KUKA KRL program: Station200_UpStacker.src, Station200_UpStacker.dat

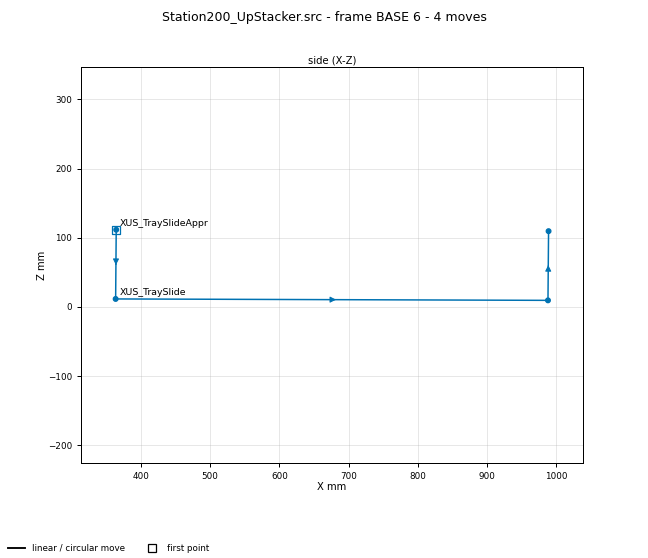
[picture p0: tool path of Station200_UpStacker.src in frame BASE 6, 4 of 12 moves have a stored position in this frame; points joined in program order, loops and branches not executed]
--- Station200_UpStacker.src ---
&ACCESS RVO1
&REL 54
&PARAM DISKPATH = KRC:\R1\Program
DEF Station200_UpStacker()

   ;FOLD INI;%{PE}
      ;FOLD BASISTECH INI
         GLOBAL INTERRUPT DECL 3 WHEN $STOPMESS == TRUE DO IR_STOPM()
         INTERRUPT ON 3
         BAS(#INITMOV, 0)
      ;ENDFOLD (BASISTECH INI)
      ;FOLD USER INI
         ;Make your modifications here
      ;ENDFOLD (USER INI)
      ;ENDFOLD (INI)

      PickPlaceTrayTeach()

;FOLD SPTP US_A1Turn Vel=100 % PDAT8 Tool[0] Base[0] ;%{PE}
;FOLD Parameters ;%{h}
;Params IlfProvider=kukaroboter.basistech.inlineforms.movement.spline; Kuka.IsGlobalPoint=False; Kuka.PointName=US_A1Turn; Kuka.BlendingEnabled=False; Kuka.MoveDataPtpName=PDAT8; Kuka.VelocityPtp=100; Kuka.VelocityFieldEnabled=True; Kuka.ColDetectFieldEnabled=True; Kuka.CurrentCDSetIndex=0; Kuka.MovementParameterFieldEnabled=True; IlfCommand=SPTP
;ENDFOLD
SPTP XUS_A1Turn WITH $VEL_AXIS[1] = SVEL_JOINT(100.0), $TOOL = STOOL2(FUS_A1Turn), $BASE = SBASE(FUS_A1Turn.BASE_NO), $IPO_MODE = SIPO_MODE(FUS_A1Turn.IPO_FRAME), $LOAD = SLOAD(FUS_A1Turn.TOOL_NO), $ACC_AXIS[1] = SACC_JOINT(PPDAT8), $APO = SAPO_PTP(PPDAT8), $GEAR_JERK[1] = SGEAR_JERK(PPDAT8), $COLLMON_TOL_PRO[1] = USE_CM_PRO_VALUES(0)
;ENDFOLD

;If tray layer needs to be moved, move layer before anything else happens.
If UStoR_ReqToMoveLayer==True Then
;FOLD SPTP US_TraySlideAppr Vel=100 % PDAT9 Tool[3]:TraySlidePin Base[6]:StackerFrame ;%{PE}
;FOLD Parameters ;%{h}
;Params IlfProvider=kukaroboter.basistech.inlineforms.movement.spline; Kuka.IsGlobalPoint=False; Kuka.PointName=US_TraySlideAppr; Kuka.BlendingEnabled=False; Kuka.MoveDataPtpName=PDAT9; Kuka.VelocityPtp=100; Kuka.VelocityFieldEnabled=True; Kuka.ColDetectFieldEnabled=True; Kuka.CurrentCDSetIndex=0; Kuka.MovementParameterFieldEnabled=True; IlfCommand=SPTP
;ENDFOLD
SPTP XUS_TraySlideAppr WITH $VEL_AXIS[1] = SVEL_JOINT(100.0), $TOOL = STOOL2(FUS_TraySlideAppr), $BASE = SBASE(FUS_TraySlideAppr.BASE_NO), $IPO_MODE = SIPO_MODE(FUS_TraySlideAppr.IPO_FRAME), $LOAD = SLOAD(FUS_TraySlideAppr.TOOL_NO), $ACC_AXIS[1] = SACC_JOINT(PPDAT9), $APO = SAPO_PTP(PPDAT9), $GEAR_JERK[1] = SGEAR_JERK(PPDAT9), $COLLMON_TOL_PRO[1] = USE_CM_PRO_VALUES(0)
;ENDFOLD
;FOLD SLIN US_TraySlide Vel=0.2 m/s CPDAT07 Tool[3]:TraySlidePin Base[6]:StackerFrame ;%{PE}
;FOLD Parameters ;%{h}
;Params IlfProvider=kukaroboter.basistech.inlineforms.movement.spline; Kuka.IsGlobalPoint=False; Kuka.PointName=US_TraySlide; Kuka.BlendingEnabled=False; Kuka.MoveDataName=CPDAT07; Kuka.VelocityPath=0.2; Kuka.VelocityFieldEnabled=True; Kuka.ColDetectFieldEnabled=True; Kuka.CurrentCDSetIndex=0; Kuka.MovementParameterFieldEnabled=True; IlfCommand=SLIN
;ENDFOLD
SLIN XUS_TraySlide WITH $VEL = SVEL_CP(0.2, , LCPDAT07), $TOOL = STOOL2(FUS_TraySlide), $BASE = SBASE(FUS_TraySlide.BASE_NO), $IPO_MODE = SIPO_MODE(FUS_TraySlide.IPO_FRAME), $LOAD = SLOAD(FUS_TraySlide.TOOL_NO), $ACC = SACC_CP(LCPDAT07), $ORI_TYPE = SORI_TYP(LCPDAT07), $APO = SAPO(LCPDAT07), $JERK = SJERK(LCPDAT07), $COLLMON_TOL_PRO[1] = USE_CM_PRO_VALUES(0)
;ENDFOLD
;FOLD SLIN US_TraySlideEnd Vel=0.15 m/s CPDAT08 Tool[3]:TraySlidePin Base[6]:StackerFrame ;%{PE}
;FOLD Parameters ;%{h}
;Params IlfProvider=kukaroboter.basistech.inlineforms.movement.spline; Kuka.IsGlobalPoint=False; Kuka.PointName=US_TraySlideEnd; Kuka.BlendingEnabled=False; Kuka.MoveDataName=CPDAT08; Kuka.VelocityPath=0.15; Kuka.VelocityFieldEnabled=True; Kuka.ColDetectFieldEnabled=True; Kuka.CurrentCDSetIndex=0; Kuka.MovementParameterFieldEnabled=True; IlfCommand=SLIN
;ENDFOLD
SLIN XUS_TraySlideEnd WITH $VEL = SVEL_CP(0.15, , LCPDAT08), $TOOL = STOOL2(FUS_TraySlideEnd), $BASE = SBASE(FUS_TraySlideEnd.BASE_NO), $IPO_MODE = SIPO_MODE(FUS_TraySlideEnd.IPO_FRAME), $LOAD = SLOAD(FUS_TraySlideEnd.TOOL_NO), $ACC = SACC_CP(LCPDAT08), $ORI_TYPE = SORI_TYP(LCPDAT08), $APO = SAPO(LCPDAT08), $JERK = SJERK(LCPDAT08), $COLLMON_TOL_PRO[1] = USE_CM_PRO_VALUES(0)
;ENDFOLD
;FOLD SLIN US_TraySlideReturn Vel=0.2 m/s CPDAT09 Tool[3]:TraySlidePin Base[6]:StackerFrame ;%{PE}
;FOLD Parameters ;%{h}
;Params IlfProvider=kukaroboter.basistech.inlineforms.movement.spline; Kuka.IsGlobalPoint=False; Kuka.PointName=US_TraySlideReturn; Kuka.BlendingEnabled=False; Kuka.MoveDataName=CPDAT09; Kuka.VelocityPath=0.2; Kuka.VelocityFieldEnabled=True; Kuka.ColDetectFieldEnabled=True; Kuka.CurrentCDSetIndex=0; Kuka.MovementParameterFieldEnabled=True; IlfCommand=SLIN
;ENDFOLD
SLIN XUS_TraySlideReturn WITH $VEL = SVEL_CP(0.2, , LCPDAT09), $TOOL = STOOL2(FUS_TraySlideReturn), $BASE = SBASE(FUS_TraySlideReturn.BASE_NO), $IPO_MODE = SIPO_MODE(FUS_TraySlideReturn.IPO_FRAME), $LOAD = SLOAD(FUS_TraySlideReturn.TOOL_NO), $ACC = SACC_CP(LCPDAT09), $ORI_TYPE = SORI_TYP(LCPDAT09), $APO = SAPO(LCPDAT09), $JERK = SJERK(LCPDAT09), $COLLMON_TOL_PRO[1] = USE_CM_PRO_VALUES(0)
;ENDFOLD
;FOLD SPTP DS_A1Turn Vel=100 % PDAT10 Tool[0] Base[0] ;%{PE}
;FOLD Parameters ;%{h}
;Params IlfProvider=kukaroboter.basistech.inlineforms.movement.spline; Kuka.IsGlobalPoint=False; Kuka.PointName=DS_A1Turn; Kuka.BlendingEnabled=False; Kuka.MoveDataPtpName=PDAT10; Kuka.VelocityPtp=100; Kuka.VelocityFieldEnabled=True; Kuka.ColDetectFieldEnabled=True; Kuka.CurrentCDSetIndex=0; Kuka.MovementParameterFieldEnabled=True; IlfCommand=SPTP
;ENDFOLD
SPTP XDS_A1Turn WITH $VEL_AXIS[1] = SVEL_JOINT(100.0), $TOOL = STOOL2(FDS_A1Turn), $BASE = SBASE(FDS_A1Turn.BASE_NO), $IPO_MODE = SIPO_MODE(FDS_A1Turn.IPO_FRAME), $LOAD = SLOAD(FDS_A1Turn.TOOL_NO), $ACC_AXIS[1] = SACC_JOINT(PPDAT10), $APO = SAPO_PTP(PPDAT10), $GEAR_JERK[1] = SGEAR_JERK(PPDAT10), $COLLMON_TOL_PRO[1] = USE_CM_PRO_VALUES(0)
;ENDFOLD
       RtoUS_LayerMovedConfirm=True
       wait sec .1
       RtoUS_LayerMovedConfirm=False
GOTO EndOfModule
EndIf


;Clear vacuum cups outputs
RtoPLC_BlankCupAVac=False
RtoPLC_BlankCupBVac=False
RtoPLC_BlankCupABlow=False
RtoPLC_BlankCupBBlow=False
RtoUS_PickConfirm=False
RobotCell_Error=False

;Check for layer mover, if needed slide upstacker tray to downstacker



 ;move tooling to row and column approach position for pick, then slowy move into the pick position
            US_PickApproach[UStoR_PickRowNumber,UStoR_PickColumnNumber] = US_Pick[UStoR_PickRowNumber,UStoR_PickColumnNumber]
            US_PickApproach[UStoR_PickRowNumber,UStoR_PickColumnNumber].Z = US_PickApproach[UStoR_PickRowNumber,UStoR_PickColumnNumber].Z + 100
            US_PickApproachSlow[UStoR_PickRowNumber,UStoR_PickColumnNumber].Z = US_PickApproach[UStoR_PickRowNumber,UStoR_PickColumnNumber].Z - 65


 SPTP US_PickApproach[UStoR_PickRowNumber,UStoR_PickColumnNumber] with $TOOL=TOOL_DATA[1],$BASE=BASE_DATA[1],$LOAD=LOAD_DATA[1],$VEL.CP = 2
 SLIN US_PickApproachSlow[UStoR_PickRowNumber,UStoR_PickColumnNumber] with $TOOL=TOOL_DATA[1],$BASE=BASE_DATA[1],$LOAD=LOAD_DATA[1],$VEL.CP = 2
 SLIN US_Pick[UStoR_PickRowNumber,UStoR_PickColumnNumber] with $TOOL=TOOL_DATA[1],$BASE=BASE_DATA[1],$LOAD=LOAD_DATA[1],$VEL.CP = 0.1

;Set vacuum cups to on
RtoPLC_BlankCupAVac=True
RtoPLC_BlankCupBVac=True

      $TIMER_STOP[2]=True ;stop timer
       $TIMER[2]=0 ;reset timer
       $TIMER_STOP[2]=False ;stop timer
       Loop
       If (($TIMER[2]>=5000) Or ((PLCtoR_BlankCupAVacOn==True) And (PLCtoR_BlankCupBVacOn==True)))Then
              $TIMER_STOP[2]=True ;stop timer
              $TIMER[2]=0 ;reset time
             Exit
endif
         EndLoop
;check vacuum sensors for being false, if false, set suction cup error bits
If ((PLCtoR_BlankCupAVacOn==False) Or (PLCtoR_BlankCupBVacOn==False)) Then

       If PLCtoR_BlankCupAVacOn==False Then
              RtoUS_PickErrorVG524=True

       EndIf
       If PLCtoR_BlankCupBVacOn==False Then
              RtoUS_PickErrorVG526=True

       EndIf
EndIf

;check if vacuum error bits were set, if set, turn off vacuum cups, blow off, reset error bits
If ((RtoUS_PickErrorVG524==True) Or (RtoUS_PickErrorVG526==True)) Then
       Wait Sec .25
       RtoPLC_BlankCupAVac=False
       RtoPLC_BlankCupBVac=False
       RtoPLC_BlankCupABlow=True
       RtoPLC_BlankCupBBlow=True
       Wait Sec .25
       RtoPLC_BlankCupABlow=False
       RtoPLC_BlankCupBBlow=False
       RtoUS_PickErrorVG524=False
       RtoUS_PickErrorVG526=False

       SLIN US_PickApproach[UStoR_PickRowNumber,UStoR_PickColumnNumber] with $TOOL=TOOL_DATA[1],$BASE=BASE_DATA[1],$LOAD=LOAD_DATA[1],$VEL.CP = 2
EndIf

;check vacuum sensors for being true, if true, slowly lift parts from tray
If ((PLCtoR_BlankCupAVacOn==True) And (PLCtoR_BlankCupBVacOn==True)) Then
       SLIN US_PickApproach[UStoR_PickRowNumber,UStoR_PickColumnNumber] with $TOOL=TOOL_DATA[1],$BASE=BASE_DATA[1],$LOAD=LOAD_DATA[1],$VEL.CP = 2
EndIf


;FOLD SPTP US_A1Return Vel=100 % PDAT4 Tool[0] Base[0] ;%{PE}
;FOLD Parameters ;%{h}
;Params IlfProvider=kukaroboter.basistech.inlineforms.movement.spline; Kuka.IsGlobalPoint=False; Kuka.PointName=US_A1Return; Kuka.BlendingEnabled=False; Kuka.MoveDataPtpName=PDAT4; Kuka.VelocityPtp=100; Kuka.VelocityFieldEnabled=True; Kuka.ColDetectFieldEnabled=True; Kuka.CurrentCDSetIndex=0; Kuka.MovementParameterFieldEnabled=True; IlfCommand=SPTP
;ENDFOLD
SPTP XUS_A1Return WITH $VEL_AXIS[1] = SVEL_JOINT(100.0), $TOOL = STOOL2(FUS_A1Return), $BASE = SBASE(FUS_A1Return.BASE_NO), $IPO_MODE = SIPO_MODE(FUS_A1Return.IPO_FRAME), $LOAD = SLOAD(FUS_A1Return.TOOL_NO), $ACC_AXIS[1] = SACC_JOINT(PPDAT4), $APO = SAPO_PTP(PPDAT4), $GEAR_JERK[1] = SGEAR_JERK(PPDAT4), $COLLMON_TOL_PRO[1] = USE_CM_PRO_VALUES(0)
;ENDFOLD

;check vacuum sensors again for being false, if false, set suction cup error bits
If ((PLCtoR_BlankCupAVacOn==False) Or (PLCtoR_BlankCupBVacOn==False)) Then
       Wait Sec 2
       If PLCtoR_BlankCupAVacOn==False Then
              RtoUS_PickErrorVG524=True

       EndIf
       If PLCtoR_BlankCupBVacOn==False Then
              RtoUS_PickErrorVG526=True

       EndIf
EndIf

;check vacuum sensors again for being true, if true, set pick confirm bit for .5 seconds, copy sequence number to tool, set tooling has-parts bit,  END this module program
If ((PLCtoR_BlankCupAVacOn==True) And (PLCtoR_BlankCupBVacOn==True)) Then
       RtoPLC_ToolBlnkSeqNumber=UStoR_PickSeqNumber
       RtoUS_PickConfirm=True
       Wait Sec .25
       RtoUS_PickConfirm=False
       RtoPLC_ToolBlnkHasParts=True

EndIf

;check again if vacuum error bits were set, if set, turn off vacuum cups, blow off, reset error bits, set tooling has-parts bit, call reject blanks module program
If ((RtoUS_PickErrorVG524==True) Or (RtoUS_PickErrorVG526==True)) Then
       Wait Sec .25
       RtoUS_PickErrorVG524=False
       RtoUS_PickErrorVG526=False
       RtoPLC_ToolBlnkHasParts=True
       Rjct_1Blnk_2Fin_3Both=1
       Station500_Reject()
EndIf


EndOfModule:
END

--- Station200_UpStacker.dat ---
&ACCESS RVP1
&REL 55
&PARAM DISKPATH = KRC:\R1\Program
DEFDAT  STATION200_UPSTACKER
;FOLD EXTERNAL DECLARATIONS;%{PE}%MKUKATPBASIS,%CEXT,%VCOMMON,%P
;FOLD BASISTECH EXT;%{PE}%MKUKATPBASIS,%CEXT,%VEXT,%P
EXT  BAS (BAS_COMMAND  :IN,REAL  :IN )
DECL INT SUCCESS
;ENDFOLD (BASISTECH EXT)
;FOLD USER EXT;%{E}%MKUKATPUSER,%CEXT,%VEXT,%P
;Make your modifications here

;ENDFOLD (USER EXT)
;ENDFOLD (EXTERNAL DECLARATIONS)


DECL LDAT LCPDAT1={VEL 2.00000,ACC 60.0000,APO_DIST 500.000,APO_FAC 50.0000,AXIS_VEL 100.000,AXIS_ACC 60.0000,ORI_TYP #VAR,CIRC_TYP #BASE,JERK_FAC 50.0000,GEAR_JERK 100.000,EXAX_IGN 0}
DECL PDAT PDEFAULT={VEL 100.000,ACC 60.0000,APO_DIST 500.000,APO_MODE #CDIS,GEAR_JERK 100.000,EXAX_IGN 0}
DECL LDAT LCPDAT2={VEL 2.00000,ACC 60.0000,APO_DIST 500.000,APO_FAC 50.0000,AXIS_VEL 100.000,AXIS_ACC 60.0000,ORI_TYP #VAR,CIRC_TYP #BASE,JERK_FAC 50.0000,GEAR_JERK 100.000,EXAX_IGN 0}
DECL PDAT PPDAT1={VEL 100.000,ACC 60.0000,APO_DIST 500.000,APO_MODE #CDIS,GEAR_JERK 100.000,EXAX_IGN 0}
DECL LDAT LCPDAT3={VEL 2.00000,ACC 60.0000,APO_DIST 500.000,APO_FAC 50.0000,AXIS_VEL 100.000,AXIS_ACC 60.0000,ORI_TYP #VAR,CIRC_TYP #BASE,JERK_FAC 50.0000,GEAR_JERK 100.000,EXAX_IGN 0}
DECL LDAT LCPDAT4={VEL 2.00000,ACC 60.0000,APO_DIST 500.000,APO_FAC 50.0000,AXIS_VEL 100.000,AXIS_ACC 60.0000,ORI_TYP #VAR,CIRC_TYP #BASE,JERK_FAC 50.0000,GEAR_JERK 100.000,EXAX_IGN 0}
DECL LDAT LCPDAT5={VEL 2.00000,ACC 60.0000,APO_DIST 500.000,APO_FAC 50.0000,AXIS_VEL 100.000,AXIS_ACC 60.0000,ORI_TYP #VAR,CIRC_TYP #BASE,JERK_FAC 50.0000,GEAR_JERK 100.000,EXAX_IGN 0}
DECL PDAT PPDAT2={VEL 100.000,ACC 60.0000,APO_DIST 500.000,APO_MODE #CDIS,GEAR_JERK 100.000,EXAX_IGN 0}
DECL PDAT PPDAT3={VEL 100.000,ACC 60.0000,APO_DIST 500.000,APO_MODE #CDIS,GEAR_JERK 100.000,EXAX_IGN 0}
DECL PDAT PPDAT4={VEL 100.000,ACC 60.0000,APO_DIST 500.000,APO_MODE #CDIS,GEAR_JERK 100.000,EXAX_IGN 0}
DECL E6POS XUS_A1Turn={X -108.546844,Y -232.779465,Z 1087.90991,A 64.9999619,B 35.0000,C 179.999985,S 2,T 34,E1 0.0,E2 0.0,E3 0.0,E4 0.0,E5 0.0,E6 0.0}
DECL FDAT FUS_A1Turn={TOOL_NO 0,BASE_NO 0,IPO_FRAME #BASE,POINT2[] " "}
DECL E6POS XUS_A1Return={X -108.546844,Y -232.779465,Z 1087.90991,A 64.9999619,B 35.0000,C 179.999985,S 2,T 34,E1 0.0,E2 0.0,E3 0.0,E4 0.0,E5 0.0,E6 0.0}
DECL FDAT FUS_A1Return={TOOL_NO 0,BASE_NO 0,IPO_FRAME #BASE,POINT2[] " "}
DECL LDAT LCPDAT6={VEL 2.00000,ACC 60.0000,APO_DIST 500.000,APO_FAC 50.0000,AXIS_VEL 100.000,AXIS_ACC 60.0000,ORI_TYP #VAR,CIRC_TYP #BASE,JERK_FAC 50.0000,GEAR_JERK 100.000,EXAX_IGN 0}
DECL LDAT LCPDAT7={VEL 2.00000,ACC 60.0000,APO_DIST 500.000,APO_FAC 50.0000,AXIS_VEL 100.000,AXIS_ACC 60.0000,ORI_TYP #VAR,CIRC_TYP #BASE,JERK_FAC 50.0000,GEAR_JERK 100.000,EXAX_IGN 0}
DECL LDAT LCPDAT8={VEL 0.200000,ACC 60.0000,APO_DIST 500.000,APO_FAC 50.0000,AXIS_VEL 100.000,AXIS_ACC 60.0000,ORI_TYP #VAR,CIRC_TYP #BASE,JERK_FAC 50.0000,GEAR_JERK 100.000,EXAX_IGN 0}
DECL LDAT LCPDAT9={VEL 0.200000,ACC 60.0000,APO_DIST 500.000,APO_FAC 50.0000,AXIS_VEL 100.000,AXIS_ACC 60.0000,ORI_TYP #VAR,CIRC_TYP #BASE,JERK_FAC 50.0000,GEAR_JERK 100.000,EXAX_IGN 0}
DECL LDAT LCPDAT10={VEL 0.200000,ACC 60.0000,APO_DIST 500.000,APO_FAC 50.0000,AXIS_VEL 100.000,AXIS_ACC 60.0000,ORI_TYP #VAR,CIRC_TYP #BASE,JERK_FAC 50.0000,GEAR_JERK 100.000,EXAX_IGN 0}
DECL E6POS XUS_TraySlideAppr={X 364.230621,Y 241.480240,Z 111.502525,A -0.00475764973,B 0.488523424,C -0.0135169579,S 2,T 2,E1 0.0,E2 0.0,E3 0.0,E4 0.0,E5 0.0,E6 0.0}
DECL FDAT FUS_TraySlideAppr={TOOL_NO 3,BASE_NO 6,IPO_FRAME #BASE,POINT2[] " "}
DECL E6POS XUS_TraySlide={X 363.377350,Y 241.456268,Z 11.5069418,A -0.00488120038,B 0.488478780,C -0.0135536417,S 2,T 10,E1 0.0,E2 0.0,E3 0.0,E4 0.0,E5 0.0,E6 0.0}
DECL FDAT FUS_TraySlide={TOOL_NO 3,BASE_NO 6,IPO_FRAME #BASE,POINT2[] " "}
DECL E6POS XUS_TraySlideReturn={X 989.015259,Y 242.827,Z 109.465332,A -0.00488119852,B 0.488478750,C -0.0135536510,S 2,T 2,E1 0.0,E2 0.0,E3 0.0,E4 0.0,E5 0.0,E6 0.0}
DECL FDAT FUS_TraySlideReturn={TOOL_NO 3,BASE_NO 6,IPO_FRAME #BASE,POINT2[] " "}
DECL E6POS XUS_TraySlideEnd={X 988.162720,Y 242.803406,Z 9.46896839,A -0.00488119433,B 0.488478750,C -0.0135536417,S 2,T 2,E1 0.0,E2 0.0,E3 0.0,E4 0.0,E5 0.0,E6 0.0}
DECL FDAT FUS_TraySlideEnd={TOOL_NO 3,BASE_NO 6,IPO_FRAME #BASE,POINT2[] " "}
DECL PDAT PPDAT5={VEL 100.000,ACC 60.0000,APO_DIST 500.000,APO_MODE #CDIS,GEAR_JERK 100.000,EXAX_IGN 0}
DECL E6POS XDS_A1Turn={X 44.6004448,Y -252.941681,Z 1087.90991,A 99.9999619,B 35.0000,C 179.999985,S 2,T 34,E1 0.0,E2 0.0,E3 0.0,E4 0.0,E5 0.0,E6 0.0}
DECL FDAT FDS_A1Turn={TOOL_NO 0,BASE_NO 0,IPO_FRAME #BASE,POINT2[] " "}

DECL PDAT PPDAT11={VEL 100.000,ACC 60.0000,APO_DIST 500.000,APO_MODE #CDIS,GEAR_JERK 100.000,EXAX_IGN 0}



DECL PDAT PPDAT6={VEL 100.000,ACC 60.0000,APO_DIST 500.000,APO_MODE #CDIS,GEAR_JERK 100.000,EXAX_IGN 0}
DECL MODULEPARAM_T LAST_TP_PARAMS={PARAMS[] "Kuka.VelocityFieldEnabled=True; Kuka.ColDetectFieldEnabled=True; Kuka.MovementParameterFieldEnabled=True; Kuka.IsAngleEnabled=False; Kuka.PointName=US_TraySlideEnd; Kuka.FrameData.base_no=6; Kuka.FrameData.tool_no=3; Kuka.FrameData.ipo_frame=#BASE; Kuka.isglobalpoint=False; Kuka.MoveDataPtpName=PDAT4; Kuka.MovementDataPdat.apo_mode=#CDIS; Kuka.MovementDataPdat.apo_dist=500; Kuka.MovementData.vel=0.15; Kuka.MovementData.acc=10; Kuka.MovementData.exax_ign=0; Kuka.VelocityPtp=100; Kuka.BlendingEnabled=False; Kuka.APXEnabled=False; Kuka.CurrentCDSetIndex=0; Kuka.FrameData.point2=; Kuka.MoveDataName=CPDAT08; Kuka.MovementData.cb={AUX_PT {ORI #CONSIDER,E1 #CONSIDER,E2 #CONSIDER,E3 #CONSIDER,E4 #CONSIDER,E5 #CONSIDER,E6 #CONSIDER},TARGET_PT {ORI #INTERPOLATE,E1 #INTERPOLATE,E2 #INTERPOLATE,E3 #INTERPOLATE,E4 #INTERPOLATE,E5 #INTERPOLATE,E6 #INTERPOLATE}}; Kuka.MovementData.apo_fac=50; Kuka.MovementData.apo_dist=500; Kuka.MovementData.axis_acc=60; Kuka.MovementData.axis_vel=100; Kuka.MovementData.circ_typ=#BASE; Kuka.MovementData.jerk_fac=50; Kuka.MovementData.ori_typ=#VAR; Kuka.VelocityPath=0.15   "}
DECL PDAT PPDAT7={VEL 100.000,ACC 60.0000,APO_DIST 500.000,APO_MODE #CDIS,GEAR_JERK 100.000,EXAX_IGN 0}
DECL FDAT FUS_TeachPick={TOOL_NO 1,BASE_NO 1,IPO_FRAME #BASE,POINT2[] " "}
DECL E6POS XUS_TeachPick={X 0.936865628,Y 182.409576,Z 5.05940,A 90.0592346,B 1.36682522,C 179.845459,S 2,T 34,E1 0.0,E2 0.0,E3 0.0,E4 0.0,E5 0.0,E6 0.0}
DECL LDAT LCPDAT01={VEL 2.00000,ACC 60.0000,APO_DIST 500.000,APO_FAC 50.0000,AXIS_VEL 100.000,AXIS_ACC 60.0000,ORI_TYP #VAR,CIRC_TYP #BASE,JERK_FAC 50.0000,GEAR_JERK 100.000,EXAX_IGN 0,CB {AUX_PT {ORI #CONSIDER,E1 #CONSIDER,E2 #CONSIDER,E3 #CONSIDER,E4 #CONSIDER,E5 #CONSIDER,E6 #CONSIDER},TARGET_PT {ORI #INTERPOLATE,E1 #INTERPOLATE,E2 #INTERPOLATE,E3 #INTERPOLATE,E4 #INTERPOLATE,E5 #INTERPOLATE,E6 #INTERPOLATE}}}
DECL E6POS US_PickApproach_1[2,4]
DECL E6POS US_PickApproachSlow_1[1,1]
DECL LDAT LCPDAT02={VEL 0.200000,ACC 60.0000,APO_DIST 500.000,APO_FAC 50.0000,AXIS_VEL 100.000,AXIS_ACC 60.0000,ORI_TYP #VAR,CIRC_TYP #BASE,JERK_FAC 50.0000,GEAR_JERK 100.000,EXAX_IGN 0,CB {AUX_PT {ORI #CONSIDER,E1 #CONSIDER,E2 #CONSIDER,E3 #CONSIDER,E4 #CONSIDER,E5 #CONSIDER,E6 #CONSIDER},TARGET_PT {ORI #INTERPOLATE,E1 #INTERPOLATE,E2 #INTERPOLATE,E3 #INTERPOLATE,E4 #INTERPOLATE,E5 #INTERPOLATE,E6 #INTERPOLATE}}}
DECL LDAT LCPDAT03={VEL 0.200000,ACC 60.0000,APO_DIST 500.000,APO_FAC 50.0000,AXIS_VEL 100.000,AXIS_ACC 60.0000,ORI_TYP #VAR,CIRC_TYP #BASE,JERK_FAC 50.0000,GEAR_JERK 100.000,EXAX_IGN 0,CB {AUX_PT {ORI #CONSIDER,E1 #CONSIDER,E2 #CONSIDER,E3 #CONSIDER,E4 #CONSIDER,E5 #CONSIDER,E6 #CONSIDER},TARGET_PT {ORI #INTERPOLATE,E1 #INTERPOLATE,E2 #INTERPOLATE,E3 #INTERPOLATE,E4 #INTERPOLATE,E5 #INTERPOLATE,E6 #INTERPOLATE}}}
DECL E6POS XUS_TeachPick1={X 0.927678406,Y 183.215424,Z 5.87333918,A 90.0619583,B 0.366831064,C 179.842010,S 2,T 34,E1 0.0,E2 0.0,E3 0.0,E4 0.0,E5 0.0,E6 0.0}
DECL FDAT FUS_TeachPick1={TOOL_NO 1,BASE_NO 1,IPO_FRAME #BASE,POINT2[] " "}
DECL LDAT LCPDAT04={VEL 1.00000,ACC 60.0000,APO_DIST 500.000,APO_FAC 50.0000,AXIS_VEL 100.000,AXIS_ACC 60.0000,ORI_TYP #VAR,CIRC_TYP #BASE,JERK_FAC 50.0000,GEAR_JERK 100.000,EXAX_IGN 0,CB {AUX_PT {ORI #CONSIDER,E1 #CONSIDER,E2 #CONSIDER,E3 #CONSIDER,E4 #CONSIDER,E5 #CONSIDER,E6 #CONSIDER},TARGET_PT {ORI #INTERPOLATE,E1 #INTERPOLATE,E2 #INTERPOLATE,E3 #INTERPOLATE,E4 #INTERPOLATE,E5 #INTERPOLATE,E6 #INTERPOLATE}}}
DECL E6POS XUS_TeachPick2={X 2.76713896,Y 182.527664,Z 5.28286,A 90.0619583,B 0.366831064,C 179.842010,S 2,T 34,E1 0.0,E2 0.0,E3 0.0,E4 0.0,E5 0.0,E6 0.0}
DECL FDAT FUS_TeachPick2={TOOL_NO 1,BASE_NO 1,IPO_FRAME #BASE,POINT2[] " "}
DECL LDAT LCPDAT05={VEL 1.00000,ACC 60.0000,APO_DIST 500.000,APO_FAC 50.0000,AXIS_VEL 100.000,AXIS_ACC 60.0000,ORI_TYP #VAR,CIRC_TYP #BASE,JERK_FAC 50.0000,GEAR_JERK 100.000,EXAX_IGN 0,CB {AUX_PT {ORI #CONSIDER,E1 #CONSIDER,E2 #CONSIDER,E3 #CONSIDER,E4 #CONSIDER,E5 #CONSIDER,E6 #CONSIDER},TARGET_PT {ORI #INTERPOLATE,E1 #INTERPOLATE,E2 #INTERPOLATE,E3 #INTERPOLATE,E4 #INTERPOLATE,E5 #INTERPOLATE,E6 #INTERPOLATE}}}
DECL E6POS XUS_TeachPick3={X 0.172189355,Y 180.890,Z 4.88615656,A 90.0619583,B 0.366835088,C 179.842010,S 2,T 34,E1 0.0,E2 0.0,E3 0.0,E4 0.0,E5 0.0,E6 0.0}
DECL FDAT FUS_TeachPick3={TOOL_NO 1,BASE_NO 1,IPO_FRAME #BASE,POINT2[] " "}
DECL LDAT LCPDAT06={VEL 1.00000,ACC 60.0000,APO_DIST 500.000,APO_FAC 50.0000,AXIS_VEL 100.000,AXIS_ACC 60.0000,ORI_TYP #VAR,CIRC_TYP #BASE,JERK_FAC 50.0000,GEAR_JERK 100.000,EXAX_IGN 0,CB {AUX_PT {ORI #CONSIDER,E1 #CONSIDER,E2 #CONSIDER,E3 #CONSIDER,E4 #CONSIDER,E5 #CONSIDER,E6 #CONSIDER},TARGET_PT {ORI #INTERPOLATE,E1 #INTERPOLATE,E2 #INTERPOLATE,E3 #INTERPOLATE,E4 #INTERPOLATE,E5 #INTERPOLATE,E6 #INTERPOLATE}}}
DECL PDAT PPDAT8={VEL 100.000,ACC 100.000,APO_DIST 500.000,APO_MODE #CDIS,GEAR_JERK 100.000,EXAX_IGN 0}
DECL PDAT PPDAT9={VEL 100.000,ACC 100.000,APO_DIST 500.000,APO_MODE #CDIS,GEAR_JERK 100.000,EXAX_IGN 0}
DECL LDAT LCPDAT07={VEL 0.200000,ACC 10.0000,APO_DIST 500.000,APO_FAC 50.0000,AXIS_VEL 100.000,AXIS_ACC 60.0000,ORI_TYP #VAR,CIRC_TYP #BASE,JERK_FAC 50.0000,GEAR_JERK 100.000,EXAX_IGN 0,CB {AUX_PT {ORI #CONSIDER,E1 #CONSIDER,E2 #CONSIDER,E3 #CONSIDER,E4 #CONSIDER,E5 #CONSIDER,E6 #CONSIDER},TARGET_PT {ORI #INTERPOLATE,E1 #INTERPOLATE,E2 #INTERPOLATE,E3 #INTERPOLATE,E4 #INTERPOLATE,E5 #INTERPOLATE,E6 #INTERPOLATE}}}
DECL LDAT LCPDAT08={VEL 0.150000,ACC 10.0000,APO_DIST 500.000,APO_FAC 50.0000,AXIS_VEL 100.000,AXIS_ACC 60.0000,ORI_TYP #VAR,CIRC_TYP #BASE,JERK_FAC 50.0000,GEAR_JERK 100.000,EXAX_IGN 0,CB {AUX_PT {ORI #CONSIDER,E1 #CONSIDER,E2 #CONSIDER,E3 #CONSIDER,E4 #CONSIDER,E5 #CONSIDER,E6 #CONSIDER},TARGET_PT {ORI #INTERPOLATE,E1 #INTERPOLATE,E2 #INTERPOLATE,E3 #INTERPOLATE,E4 #INTERPOLATE,E5 #INTERPOLATE,E6 #INTERPOLATE}}}
DECL LDAT LCPDAT09={VEL 0.200000,ACC 60.0000,APO_DIST 500.000,APO_FAC 50.0000,AXIS_VEL 100.000,AXIS_ACC 60.0000,ORI_TYP #VAR,CIRC_TYP #BASE,JERK_FAC 50.0000,GEAR_JERK 100.000,EXAX_IGN 0,CB {AUX_PT {ORI #CONSIDER,E1 #CONSIDER,E2 #CONSIDER,E3 #CONSIDER,E4 #CONSIDER,E5 #CONSIDER,E6 #CONSIDER},TARGET_PT {ORI #INTERPOLATE,E1 #INTERPOLATE,E2 #INTERPOLATE,E3 #INTERPOLATE,E4 #INTERPOLATE,E5 #INTERPOLATE,E6 #INTERPOLATE}}}
DECL PDAT PPDAT10={VEL 100.000,ACC 60.0000,APO_DIST 500.000,APO_MODE #CDIS,GEAR_JERK 100.000,EXAX_IGN 0}
ENDDAT
